FUNCTION_BLOCK fCnt
VAR_INPUT
	///Valor contador
	iCnt: UDINT;
END_VAR

(*Entrada tipo 1008 BECHOFF CNT*)

END_FUNCTION_BLOCK

(* stored: Version 1.1.0.1, ProductVersion 3.1.4024.10
   POU fCnt: Id {ed3495eb-2095-47cc-ac62-b769e279df5e}, SpecialFunc None *)
